FUNCTION FC_KeepBetweenMinMax : LREAL			// Keeps the given iValue in between iMin (Floor) and iMax (Ceiling)  
VAR_INPUT
	iValue:		LREAL;
	iMin:		LREAL;
	iMax:		LREAL;
END_VAR

IF (iValue > iMax) THEN
	FC_KeepBetweenMinMax := iMax;
ELSIF (iValue < iMin) THEN
	FC_KeepBetweenMinMax := iMin;
ELSE
	FC_KeepBetweenMinMax := iValue;
END_IF

END_FUNCTION

(* stored: Version 1.1.0.1, ProductVersion 3.1.4026.18
   POU FC_KeepBetweenMinMax: Id {bff08ce8-4787-448e-ace6-9056e18c7353}, SpecialFunc None *)
